Omron CX-Programmer project NewProject (CX-Programmer 9.75)

# PLC NewPLC1: CP1L M

## Global symbols (name address type ; comment)
0.00 BOOL  ; PB ON 1
0.01 BOOL  ; PB OFF 1
0.02 BOOL  ; PB ON 2
0.03 BOOL  ; PB OFF 2
100.00 BOOL  ; K1
100.01 BOOL  ; K2

## Program NewProgram1 (cyclic task 0)

### Section Section1

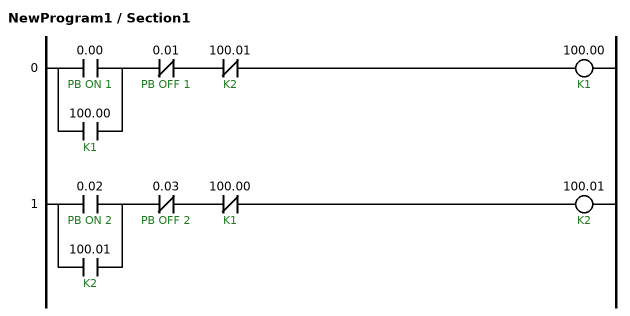
; rung 0
LD 0.00  ; PB ON 1
OR 100.00  ; K1
ANDNOT 0.01  ; PB OFF 1
ANDNOT 100.01  ; K2
OUT 100.00  ; K1
; rung 1
LD 0.02  ; PB ON 2
OR 100.01  ; K2
ANDNOT 0.03  ; PB OFF 2
ANDNOT 100.00  ; K1
OUT 100.01  ; K2

### Section END
; rung 0
END(001)